KUKA KRL program: panpick2.src, panpick2.dat

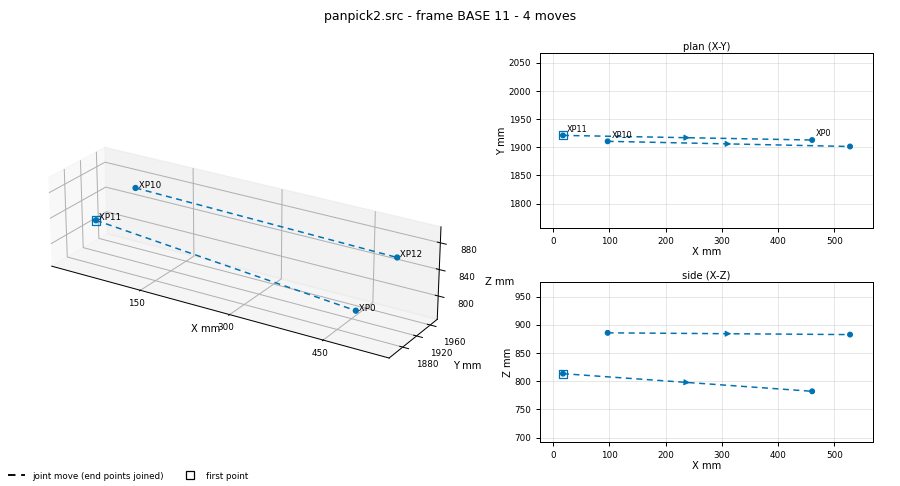
[picture p0: tool path of panpick2.src in frame BASE 11, 4 of 15 moves have a stored position in this frame; points joined in program order, loops and branches not executed]
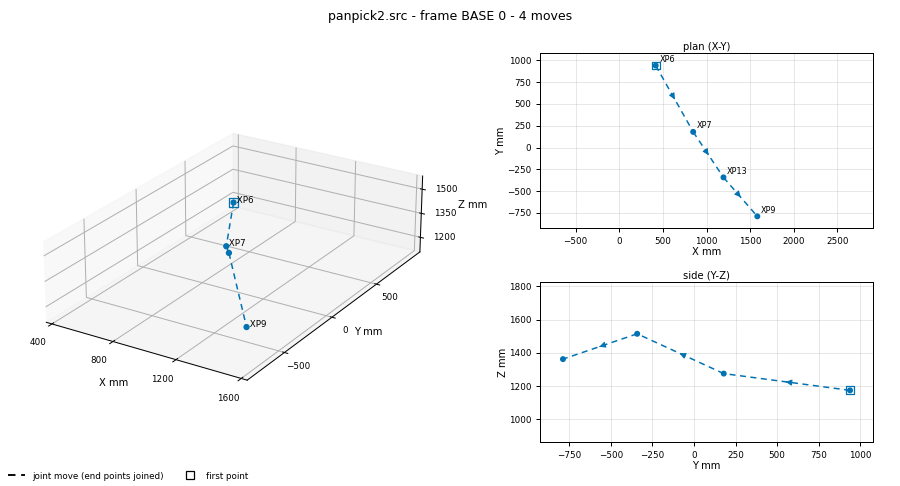
[picture p1: tool path of panpick2.src in frame BASE 0, 4 of 15 moves have a stored position in this frame; points joined in program order, loops and branches not executed]
--- panpick2.src ---
&ACCESS RVO1
&REL 4238
&PARAM EDITMASK = *
&PARAM TEMPLATE = C:\KRC\Roboter\Template\vorgabe
&PARAM DISKPATH = KRC:\R1\Program\Sub Programs
DEF panpick2( )
;FOLD INI;%{PE}
  ;FOLD BASISTECH INI
    GLOBAL INTERRUPT DECL 3 WHEN $STOPMESS==TRUE DO IR_STOPM ( )
    INTERRUPT ON 3
    BAS (#INITMOV,0 )
  ;ENDFOLD (BASISTECH INI)
  ;FOLD USER INI
    ;Make your modifications here

$ACT_BASE=0
$ACT_TOOL=0
INPICKER_Handler.DataToSend.command=0
 wait for (INPICKER_Handler.DataReceived.state==0)
;CILS_INIT()
REINTENTO=FALSE
  ;ENDFOLD (USER INI)
;ENDFOLD (INI)

xp03=$POS_ACT
PUNTOFOTO:
;POS FOTO 1
;FOLD PTP P03 CONT Vel=100 % PDAT1 Tool[0] Base[0];%{PE}%R 8.3.48,%MKUKATPBASIS,%CMOVE,%VPTP,%P 1:PTP, 2:P03, 3:C_DIS, 5:100, 7:PDAT1
$BWDSTART=FALSE
PDAT_ACT=PPDAT1
FDAT_ACT=FP03
BAS(#PTP_PARAMS,100)
PTP XP03 C_DIS
;ENDFOLD
INICIOFOTO:


;fold espera foto

 INPICKER_Handler.DataToSend.partid=0
 INPICKER_Handler.DataToSend.command=1
 wait for (INPICKER_Handler.DataReceived.state==30) or (INPICKER_Handler.dataReceived.state==-1)
 wait sec 0.5
 if (INPICKER_handler.datareceived.state==-1 )  THEN

INPICKER_Handler.DataToSend.command=0
 wait for (INPICKER_Handler.DataReceived.state==0)
goto iniciofoto
endif
;ENDFOLD
;EVALUA foto

IF (INPICKER_Handler.DataReceived.ObjectsGraspable>0)THEN

;FOLD CARGA FRAMEXP01
;FOTO OK
FRAMEAUX={X 0,Y 0,Z 0,A 0,B 0,C 0}
FRAMEAUX=INPICKER_Handler.DataReceived.PartsToGrasp0.Position
XP01.x=(FRAMEAUX.x/10)
XP01.y=(FRAMEAUX.y/10)
XP01.z=(FRAMEAUX.z/10)
XP01.a=FRAMEAUX.a/10
XP01.b=FRAMEAUX.b/10
XP01.c=FRAMEAUX.c/10
;ENDFOLD

;FOLD CARGA FRAME XP02
FRAMEAUX={X 0,Y 0,Z 0,A 0,B 0,C 0}
FRAMEAUX=INPICKER_Handler.DataReceived.PartsToGrasp0.PreGrasp0
XP02.x=(FRAMEAUX.x/10)
XP02.y=(FRAMEAUX.y/10)
XP02.z=(FRAMEAUX.z/10)
XP02.a=FRAMEAUX.a/10
XP02.b=FRAMEAUX.b/10
XP02.c=FRAMEAUX.c/10
;ENDFOLD

;FOLD Fordtech.Tool_Req Tool Request: 2 ;%{PE}%MKUKATPUSER

Tool_Req (2)

;ENDFOLD
;FOLD Fordtech.Wait_Tool_Ready Wait Tool Ready: 2 ;%{PE}%MKUKATPUSER

Wait_Tool_Ready (2)

;ENDFOLD

ELSE

IF (REINTENTO==FALSE) THEN
REINTENTO=TRUE
INPICKER_Handler.DataToSend.command=0
 wait for (INPICKER_Handler.DataReceived.state==0)
GOTO INICIOFOTO
ENDIF


;FOTO NOK
;FOLD Fordtech.Tool_Req Tool Request: 1 ;%{PE}%MKUKATPUSER

Tool_Req (1)

;ENDFOLD
;FOLD Fordtech.Wait_Tool_Ready Wait Tool Ready: 1 ;%{PE}%MKUKATPUSER

Wait_Tool_Ready (1)

;ENDFOLD

BACKJUMP=TRUE
GOTO PEXIT

ENDIF

;Baja vel si array cerca del vallado
IF (posbat==11) THEN
;FOLD PTP P11 CONT Vel=100 % M2 Tool[5] Base[11];%{PE}%R 8.3.48,%MKUKATPBASIS,%CMOVE,%VPTP,%P 1:PTP, 2:P11, 3:C_DIS, 5:100, 7:M2
$BWDSTART=FALSE
PDAT_ACT=PM2
FDAT_ACT=FP11
BAS(#PTP_PARAMS,100)
PTP XP11 C_DIS
;ENDFOLD
ACT_OV=$OV_PRO
$OV_PRO=10
ENDIF

IF (posbat==12) THEN
;FOLD PTP P0 CONT Vel=80 % M3 Tool[5] Base[11];%{PE}%R 8.3.48,%MKUKATPBASIS,%CMOVE,%VPTP,%P 1:PTP, 2:P0, 3:C_DIS, 5:80, 7:M3
$BWDSTART=FALSE
PDAT_ACT=PM3
FDAT_ACT=FP0
BAS(#PTP_PARAMS,80)
PTP XP0 C_DIS
;ENDFOLD
ACT_OV=$OV_PRO
$OV_PRO=10
ENDIF

;FOLD PTP P02 CONT Vel=100 % PDAT2 Tool[5] Base[0];%{PE}%R 8.3.48,%MKUKATPBASIS,%CMOVE,%VPTP,%P 1:PTP, 2:P02, 3:C_DIS, 5:100, 7:PDAT2
$BWDSTART=FALSE
PDAT_ACT=PPDAT2
FDAT_ACT=FP02
BAS(#PTP_PARAMS,100)
PTP XP02 C_DIS
;ENDFOLD

;FOLD LIN P01 Vel=1 m/s CPDAT3 Tool[5] Base[0];%{PE}%R 8.3.48,%MKUKATPBASIS,%CMOVE,%VLIN,%P 1:LIN, 2:P01, 3:, 5:1, 7:CPDAT3
$BWDSTART=FALSE
LDAT_ACT=LCPDAT3
FDAT_ACT=FP01
BAS(#CP_PARAMS,1)
LIN XP01
;ENDFOLD
;halt

;Cierra cilindros
CIL_BAT_ACTIVO()

;Revisa sensores y si falta alguno abre y cierra la garra 1 vez
IF NOT (($IN[243] AND $IN[244] AND $IN[245] AND $IN[247])) THEN
  $OUT[243]=TRUE
  $OUT[244]=FALSE
  WAIT SEC 0.5
  $OUT[243]=FALSE
  $OUT[244]=TRUE
ENDIF

;Mueve arriba 50mm
lin_rel {z 50}

;Revisa sensores de cilindros cerrados
;FOLD WAIT FOR ( IN 245 'CIL array closed S302B' ) CONT;%{PE}%R 8.3.48,%MKUKATPBASIS,%CEXT_WAIT_FOR,%VEXT_WAIT_FOR,%P 2:, 4:, 5:$IN, 6:245, 7:CIL array closed S302B, 9:CONTINUE
CONTINUE
WAIT FOR  ( $IN[245] )
;ENDFOLD
;FOLD WAIT FOR ( IN 247 'CIL array closed S301B' ) CONT;%{PE}%R 8.3.48,%MKUKATPBASIS,%CEXT_WAIT_FOR,%VEXT_WAIT_FOR,%P 2:, 4:, 5:$IN, 6:247, 7:CIL array closed S301B, 9:CONTINUE
CONTINUE
WAIT FOR  ( $IN[247] )
;ENDFOLD

PART_CHECK()

;FOLD WAIT FOR ( IN 257 'F carrera superior S202' );%{PE}%R 8.3.48,%MKUKATPBASIS,%CEXT_WAIT_FOR,%VEXT_WAIT_FOR,%P 2:, 4:, 5:$IN, 6:257, 7:F carrera superior S202, 9:
WAIT FOR  ( $IN[257] )
;ENDFOLD
;FOLD WAIT FOR ( IN 258 'F carrera superior S201' );%{PE}%R 8.3.48,%MKUKATPBASIS,%CEXT_WAIT_FOR,%VEXT_WAIT_FOR,%P 2:, 4:, 5:$IN, 6:258, 7:F carrera superior S201, 9:
WAIT FOR  ( $IN[258] )
;ENDFOLD


INPICKER_Handler.DataToSend.command=0

IF REINT_COGIDA==TRUE THEN
LIN_REL {Z -40}
wait sec 1
CIL_BAT_REPOSO()
PART_CHECK_OFF()
wait sec 1
LIN_REL {Z 100}
 wait for (INPICKER_Handler.DataReceived.state==0)
GOTO PUNTOFOTO
ENDIF

;Fold guardamos posicion para carton
IF (POSBAT==12) THEN
   IF ($POS_ACT.x>420) AND ($POS_ACT.x<630) THEN
      BASE_DATA[15].x=$POS_ACT.x
   ENDIF
   IF ($POS_ACT.y>1886) AND ($POS_ACT.y<2087) THEN
      BASE_DATA[15].y=$POS_ACT.y
   ENDIF
;BASE_DATA[14].z=$POS_ACT.z
ENDIF
;ENDFOLD

;fold P04

FRAMEAUX={X 0,Y 0,Z 0,A 0,B 0,C 0}
XP04=FRAMEAUX
XP04.x=XP02.x
XP04.y=XP02.y
XP04.z=(XP02.z)+110
XP04.a=XP02.a
XP04.b=XP02.b
XP04.c=XP02.c

;ENDFOLD

;FOLD PTP p04 CONT Vel=100 % PDAT4 Tool[8] Base[0];%{PE}%R 8.3.48,%MKUKATPBASIS,%CMOVE,%VPTP,%P 1:PTP, 2:p04, 3:C_DIS, 5:100, 7:PDAT4
$BWDSTART=FALSE
PDAT_ACT=PPDAT4
FDAT_ACT=Fp04
BAS(#PTP_PARAMS,100)
PTP Xp04 C_DIS
;ENDFOLD

;sube vel cuando se aleja del vallado
IF (posbat==11) THEN
;FOLD PTP P10 CONT Vel=100 % PDAT10 Tool[5] Base[11];%{PE}%R 8.3.48,%MKUKATPBASIS,%CMOVE,%VPTP,%P 1:PTP, 2:P10, 3:C_DIS, 5:100, 7:PDAT10
$BWDSTART=FALSE
PDAT_ACT=PPDAT10
FDAT_ACT=FP10
BAS(#PTP_PARAMS,100)
PTP XP10 C_DIS
;ENDFOLD
$OV_PRO=ACT_OV
ENDIF

;sube vel cuando se aleja del vallado
IF (posbat==12) THEN
;FOLD PTP P12 CONT Vel=100 % PDAT11 Tool[5] Base[11];%{PE}%R 8.3.48,%MKUKATPBASIS,%CMOVE,%VPTP,%P 1:PTP, 2:P12, 3:C_DIS, 5:100, 7:PDAT11
$BWDSTART=FALSE
PDAT_ACT=PPDAT11
FDAT_ACT=FP12
BAS(#PTP_PARAMS,100)
PTP XP12 C_DIS
;ENDFOLD
$OV_PRO=ACT_OV
ENDIF

;FOLD SYN OUT 42 'Job Ready 2' State=TRUE at START Delay=0 ms;%{PE}%R 8.3.48,%MKUKATPBASIS,%COUT,%VSYNOUT,%P 2:42, 3:Job Ready 2, 5:TRUE, 7:0, 9:0, 12:0
TRIGGER WHEN DISTANCE=0 DELAY=0 DO $OUT[42]=TRUE
;ENDFOLD
BAT_MONITOR=TRUE

;FOLD PTP P6 CONT Vel=80 % M2 Tool[8] Base[0];%{PE}%R 8.3.48,%MKUKATPBASIS,%CMOVE,%VPTP,%P 1:PTP, 2:P6, 3:C_DIS, 5:80, 7:M2
$BWDSTART=FALSE
PDAT_ACT=PM2
FDAT_ACT=FP6
BAS(#PTP_PARAMS,80)
PTP XP6 C_DIS
;ENDFOLD
;FOLD SYN OUT 18 'Area Release 2' State=TRUE at START Delay=0 ms;%{PE}%R 8.3.48,%MKUKATPBASIS,%COUT,%VSYNOUT,%P 2:18, 3:Area Release 2, 5:TRUE, 7:0, 9:0, 12:0
TRIGGER WHEN DISTANCE=0 DELAY=0 DO $OUT[18]=TRUE
;ENDFOLD
;FOLD PTP P7 CONT Vel=100 % PDAT7 Tool[8] Base[0];%{PE}%R 8.3.48,%MKUKATPBASIS,%CMOVE,%VPTP,%P 1:PTP, 2:P7, 3:C_DIS, 5:100, 7:PDAT7
$BWDSTART=FALSE
PDAT_ACT=PPDAT7
FDAT_ACT=FP7
BAS(#PTP_PARAMS,100)
PTP XP7 C_DIS
;ENDFOLD
;FOLD PTP P13 CONT Vel=100 % PDAT12 Tool[8] Base[0];%{PE}%R 8.3.48,%MKUKATPBASIS,%CMOVE,%VPTP,%P 1:PTP, 2:P13, 3:C_DIS, 5:100, 7:PDAT12
$BWDSTART=FALSE
PDAT_ACT=PPDAT12
FDAT_ACT=FP13
BAS(#PTP_PARAMS,100)
PTP XP13 C_DIS
;ENDFOLD

;FOLD PTP P9 CONT Vel=100 % PDAT9 Tool[8] Base[0];%{PE}%R 8.3.48,%MKUKATPBASIS,%CMOVE,%VPTP,%P 1:PTP, 2:P9, 3:C_DIS, 5:100, 7:PDAT9
$BWDSTART=FALSE
PDAT_ACT=PPDAT9
FDAT_ACT=FP9
BAS(#PTP_PARAMS,100)
PTP XP9 C_DIS
;ENDFOLD
PEXIT:
END

--- panpick2.dat ---
&ACCESS RVO1
&REL 4238
&PARAM EDITMASK = *
&PARAM TEMPLATE = C:\KRC\Roboter\Template\vorgabe
&PARAM DISKPATH = KRC:\R1\Program\Sub Programs
DEFDAT  panpick2
;FOLD EXTERNAL DECLARATIONS;%{PE}%MKUKATPBASIS,%CEXT,%VCOMMON,%P
;FOLD BASISTECH EXT;%{PE}%MKUKATPBASIS,%CEXT,%VEXT,%P
EXT  BAS (BAS_COMMAND  :IN,REAL  :IN )
DECL INT SUCCESS
;ENDFOLD (BASISTECH EXT)
;FOLD USER EXT;%{E}%MKUKATPUSER,%CEXT,%VEXT,%P
;Make your modifications here

;ENDFOLD (USER EXT)
;ENDFOLD (EXTERNAL DECLARATIONS)
DECL E6POS XP01={X 484.500,Y 1997.60,Z 703.400,A 271.000,B 359.900,C 180.100,S 6,T 27,E1 0.0,E2 0.0,E3 0.0,E4 0.0,E5 0.0,E6 0.0}
DECL FDAT FP01={TOOL_NO 5,BASE_NO 0,IPO_FRAME #BASE,POINT2[] " "}
DECL PDAT PPDAT01={VEL 100.000,ACC 100.000,APO_DIST 500.000,APO_MODE #CDIS,GEAR_JERK 100.000,EXAX_IGN 0}
DECL MODULEPARAM_T LAST_TP_PARAMS={PARAMS[] "Kuka.VelocityFieldEnabled=True; Kuka.ColDetectFieldEnabled=True; Kuka.MovementParameterFieldEnabled=True; Kuka.IsAngleEnabled=False; Kuka.PointName=P02; Kuka.FrameData.base_no=0; Kuka.FrameData.tool_no=5; Kuka.FrameData.ipo_frame=#BASE; Kuka.isglobalpoint=False; Kuka.MoveDataPtpName=PDAT02; Kuka.MovementDataPdat.apo_mode=#CDIS; Kuka.MovementDataPdat.apo_dist=500; Kuka.MovementData.vel=2; Kuka.MovementData.acc=100; Kuka.MovementData.exax_ign=0; Kuka.VelocityPtp=100; Kuka.BlendingEnabled=False; Kuka.APXEnabled=False; Kuka.CurrentCDSetIndex=0; Kuka.FrameData.point2=; Kuka.MoveDataName=CPDAT2; Kuka.MovementData.cb={AUX_PT {ORI #CONSIDER,E1 #CONSIDER,E2 #CONSIDER,E3 #CONSIDER,E4 #CONSIDER,E5 #CONSIDER,E6 #CONSIDER},TARGET_PT {ORI #INTERPOLATE,E1 #INTERPOLATE,E2 #INTERPOLATE,E3 #INTERPOLATE,E4 #INTERPOLATE,E5 #INTERPOLATE,E6 #INTERPOLATE}}; Kuka.MovementData.apo_fac=50; Kuka.MovementData.apo_dist=500; Kuka.MovementData.axis_acc=100; Kuka.MovementData.axis_vel=100; Kuka.MovementData.circ_typ=#BASE; Kuka.MovementData.jerk_fac=50; Kuka.MovementData.ori_typ=#VAR; Kuka.VelocityPath=2                          "}
DECL E6POS XP02={X 484.300,Y 1997.60,Z 753.400,A 271.000,B 359.900,C 180.100}
DECL FDAT FP02={TOOL_NO 5,BASE_NO 0,IPO_FRAME #BASE,POINT2[] " "}
DECL PDAT PPDAT02={VEL 100.000,ACC 100.000,APO_DIST 500.000,APO_MODE #CDIS,GEAR_JERK 100.000,EXAX_IGN 0}
DECL LDAT LCPDAT1={VEL 2.00000,ACC 100.000,APO_DIST 500.000,APO_FAC 50.0000,AXIS_VEL 100.000,AXIS_ACC 100.000,ORI_TYP #VAR,CIRC_TYP #BASE,JERK_FAC 50.0000,GEAR_JERK 100.000,EXAX_IGN 0,CB {AUX_PT {ORI #CONSIDER,E1 #CONSIDER,E2 #CONSIDER,E3 #CONSIDER,E4 #CONSIDER,E5 #CONSIDER,E6 #CONSIDER},TARGET_PT {ORI #INTERPOLATE,E1 #INTERPOLATE,E2 #INTERPOLATE,E3 #INTERPOLATE,E4 #INTERPOLATE,E5 #INTERPOLATE,E6 #INTERPOLATE}}}
DECL E6POS XP03={X 717.814697,Y 1578.53296,Z 1546.32544,A -90.8808365,B 12.0879946,C -179.654587,S 'B0110',T 'B00011011',E1 0.0,E2 0.0,E3 0.0,E4 0.0,E5 0.0,E6 0.0}
DECL FDAT FP03={TOOL_NO 0,BASE_NO 0,IPO_FRAME #BASE,POINT2[] " "}
DECL PDAT PPDAT03={VEL 100.000,ACC 100.000,APO_DIST 500.000,APO_MODE #CDIS,GEAR_JERK 100.000,EXAX_IGN 0}
DECL E6POS XP04={X 484.300,Y 1997.60,Z 863.400,A 271.000,B 359.900,C 180.100}
DECL FDAT FP04={TOOL_NO 8,BASE_NO 0,IPO_FRAME #BASE,POINT2[] " ",TQ_STATE FALSE}
DECL PDAT PPDAT04={VEL 100.000,ACC 100.000,APO_DIST 500.000,APO_MODE #CDIS,GEAR_JERK 100.000,EXAX_IGN 0}
DECL E6POS XP1={X 2856.00,Y 12860.0,Z 6727.00,A 2708.00,B 8.00000,C 1797.00}
DECL E6POS XP2={X 2856.00,Y 12860.0,Z 6727.00,A 2708.00,B 8.00000,C 1797.00}
DECL E6POS XP3={X 2856.00,Y 12860.0,Z 6727.00,A 2708.00,B 8.00000,C 1797.00}
DECL E6POS XP05={X 284.000,Y 1258.50,Z 983.400,A 271.300,B 0.800000,C 179.700,S 0,T 0,E1 0.0,E2 0.0,E3 0.0,E4 0.0,E5 0.0,E6 0.0}
DECL FDAT FP05={TOOL_NO 5,BASE_NO 0,IPO_FRAME #BASE,POINT2[] " "}
DECL PDAT PPDAT05={VEL 100.000,ACC 100.000,APO_DIST 500.000,APO_MODE #CDIS,GEAR_JERK 100.000,EXAX_IGN 0}
DECL LDAT LCPDAT2={VEL 2.00000,ACC 100.000,APO_DIST 500.000,APO_FAC 50.0000,AXIS_VEL 100.000,AXIS_ACC 100.000,ORI_TYP #VAR,CIRC_TYP #BASE,JERK_FAC 50.0000,GEAR_JERK 100.000,EXAX_IGN 0,CB {AUX_PT {ORI #CONSIDER,E1 #CONSIDER,E2 #CONSIDER,E3 #CONSIDER,E4 #CONSIDER,E5 #CONSIDER,E6 #CONSIDER},TARGET_PT {ORI #INTERPOLATE,E1 #INTERPOLATE,E2 #INTERPOLATE,E3 #INTERPOLATE,E4 #INTERPOLATE,E5 #INTERPOLATE,E6 #INTERPOLATE}}}
DECL BASIS_SUGG_T LAST_BASIS={POINT1[] "P13                     ",POINT2[] "P13                     ",CP_PARAMS[] "CPDAT0                  ",PTP_PARAMS[] "PDAT12                  ",CONT[] "C_DIS                   ",CP_VEL[] "2.0                     ",PTP_VEL[] "100                     ",SYNC_PARAMS[] "SYNCDAT                 ",SPL_NAME[] "S0                      ",A_PARAMS[] "ADAT0                   "}
DECL PDAT PPDAT1={VEL 100.000,ACC 100.000,APO_DIST 100.000,APO_MODE #CDIS,GEAR_JERK 50.0000,EXAX_IGN 0}
DECL PDAT PPDAT2={VEL 100.000,ACC 100.000,APO_DIST 100.000,APO_MODE #CDIS,GEAR_JERK 50.0000,EXAX_IGN 0}
DECL LDAT LCPDAT3={VEL 2.00000,ACC 100.000,APO_DIST 100.000,APO_FAC 50.0000,AXIS_VEL 100.000,AXIS_ACC 100.000,ORI_TYP #VAR,CIRC_TYP #BASE,JERK_FAC 50.0000,GEAR_JERK 50.0000,EXAX_IGN 0}
DECL LDAT LCPDAT4={VEL 2.00000,ACC 100.000,APO_DIST 100.000,APO_FAC 50.0000,AXIS_VEL 100.000,AXIS_ACC 100.000,ORI_TYP #VAR,CIRC_TYP #BASE,JERK_FAC 50.0000,GEAR_JERK 50.0000,EXAX_IGN 0}
DECL E6POS XP4={X 704.290344,Y 404.754028,Z 1017.77747,A -114.508537,B 15.6030617,C -167.199142,S 6,T 27,E1 0.0,E2 0.0,E3 0.0,E4 0.0,E5 0.0,E6 0.0}
DECL FDAT FP4={TOOL_NO 5,BASE_NO 0,IPO_FRAME #BASE,POINT2[] " ",TQ_STATE FALSE}
DECL PDAT PPDAT3={VEL 100.000,ACC 100.000,APO_DIST 100.000,APO_MODE #CDIS,GEAR_JERK 50.0000,EXAX_IGN 0}
DECL PDAT PPDAT4={VEL 100.000,ACC 100.000,APO_DIST 100.000,APO_MODE #CDIS,GEAR_JERK 50.0000,EXAX_IGN 0}
DECL E6POS XP5={X 1475.14294,Y -460.159363,Z 1412.20422,A -177.899490,B 3.32464623,C -176.200607,S 6,T 26,E1 0.0,E2 0.0,E3 0.0,E4 0.0,E5 0.0,E6 0.0}
DECL FDAT FP5={TOOL_NO 8,BASE_NO 0,IPO_FRAME #BASE,POINT2[] " ",TQ_STATE FALSE}
DECL PDAT PPDAT5={VEL 100.000,ACC 100.000,APO_DIST 100.000,APO_MODE #CDIS,GEAR_JERK 50.0000,EXAX_IGN 0}
DECL E6POS XP6={X 416.666626,Y 939.507,Z 1174.24280,A -97.6741943,B 4.97405386,C -178.688309,S 6,T 27,E1 0.0,E2 0.0,E3 0.0,E4 0.0,E5 0.0,E6 0.0}
DECL FDAT FP6={TOOL_NO 8,BASE_NO 0,IPO_FRAME #BASE,POINT2[] " ",TQ_STATE FALSE}
DECL PDAT PPDAT6={VEL 100.000,ACC 100.000,APO_DIST 100.000,APO_MODE #CDIS,GEAR_JERK 50.0000,EXAX_IGN 0}
DECL E6POS XP7={X 846.307739,Y 179.066498,Z 1275.12671,A -128.905045,B 18.4690285,C -164.888184,S 6,T 27,E1 0.0,E2 0.0,E3 0.0,E4 0.0,E5 0.0,E6 0.0}
DECL FDAT FP7={TOOL_NO 8,BASE_NO 0,IPO_FRAME #BASE,POINT2[] " ",TQ_STATE FALSE}
DECL PDAT PPDAT7={VEL 100.000,ACC 100.000,APO_DIST 100.000,APO_MODE #CDIS,GEAR_JERK 50.0000,EXAX_IGN 0}
DECL E6POS XP8={X 1581.36292,Y -789.059875,Z 1345.17505,A 179.845,B -0.263878196,C -172.696686,S 6,T 26,E1 0.0,E2 0.0,E3 0.0,E4 0.0,E5 0.0,E6 0.0}
DECL FDAT FP8={TOOL_NO 8,BASE_NO 0,IPO_FRAME #BASE,POINT2[] " ",TQ_STATE FALSE}
DECL PDAT PPDAT8={VEL 100.000,ACC 100.000,APO_DIST 100.000,APO_MODE #CDIS,GEAR_JERK 50.0000,EXAX_IGN 0}
DECL E6POS XP9={X 1581.36292,Y -789.059875,Z 1362.23718,A 179.674332,B -0.834132493,C -179.411911,S 6,T 26,E1 0.0,E2 0.0,E3 0.0,E4 0.0,E5 0.0,E6 0.0}
DECL FDAT FP9={TOOL_NO 8,BASE_NO 0,IPO_FRAME #BASE,POINT2[] " ",TQ_STATE FALSE}
DECL PDAT PPDAT9={VEL 100.000,ACC 100.000,APO_DIST 100.000,APO_MODE #CDIS,GEAR_JERK 50.0000,EXAX_IGN 0}
DECL E6POS XP11={X 17.7491856,Y 1921.21191,Z 813.399719,A -90.1072693,B 2.33569694,C 179.505920,S 6,T 27,E1 0.0,E2 0.0,E3 0.0,E4 0.0,E5 0.0,E6 0.0}
DECL FDAT FP11={TOOL_NO 5,BASE_NO 11,IPO_FRAME #BASE,POINT2[] " ",TQ_STATE FALSE}
DECL PDAT PM2={VEL 100.000,ACC 50.0000,APO_DIST 200.000,APO_MODE #CDIS,GEAR_JERK 50.0000,EXAX_IGN 0}
DECL PDAT PM3={VEL 100.000,ACC 50.0000,APO_DIST 200.000,APO_MODE #CDIS,GEAR_JERK 50.0000,EXAX_IGN 0}
DECL E6POS XP0={X 460.302216,Y 1912.98193,Z 782.103699,A -90.2094345,B 1.02947211,C 179.869064,S 6,T 27,E1 0.0,E2 0.0,E3 0.0,E4 0.0,E5 0.0,E6 0.0}
DECL FDAT FP0={TOOL_NO 5,BASE_NO 11,IPO_FRAME #BASE,POINT2[] " ",TQ_STATE FALSE}
DECL E6POS XP10={X 97.0999603,Y 1910.67480,Z 885.904846,A -89.8999939,B 0.400000,C 179.400,S 6,T 27,E1 0.0,E2 0.0,E3 0.0,E4 0.0,E5 0.0,E6 0.0}
DECL FDAT FP10={TOOL_NO 5,BASE_NO 11,IPO_FRAME #BASE,POINT2[] " ",TQ_STATE FALSE}
DECL PDAT PPDAT10={VEL 100.000,ACC 100.000,APO_DIST 200.000,APO_MODE #CDIS,GEAR_JERK 50.0000,EXAX_IGN 0}
DECL PDAT PPDAT11={VEL 100.000,ACC 100.000,APO_DIST 200.000,APO_MODE #CDIS,GEAR_JERK 50.0000,EXAX_IGN 0}
DECL E6POS XP12={X 527.600,Y 1901.50,Z 882.800049,A -90.1000061,B 0.200000018,C 179.900,S 6,T 27,E1 0.0,E2 0.0,E3 0.0,E4 0.0,E5 0.0,E6 0.0}
DECL FDAT FP12={TOOL_NO 5,BASE_NO 11,IPO_FRAME #BASE,POINT2[] " ",TQ_STATE FALSE}
DECL E6POS XP13={X 1193.47449,Y -342.363434,Z 1514.73352,A -173.397064,B 7.88580084,C -177.558075,S 6,T 26,E1 0.0,E2 0.0,E3 0.0,E4 0.0,E5 0.0,E6 0.0}
DECL FDAT FP13={TOOL_NO 8,BASE_NO 0,IPO_FRAME #BASE,POINT2[] " ",TQ_STATE FALSE}
DECL PDAT PPDAT12={VEL 100.000,ACC 100.000,APO_DIST 100.000,APO_MODE #CDIS,GEAR_JERK 50.0000,EXAX_IGN 0}
ENDDAT
